SYSTEM TRAFFIC_Central (* System Configuration *)
  (* Standard: 61499-1 *)
  (* Version 0.4, 2009-03-05, JHC, Holobloc Inc., Deleted Application. *)
  (* Version 0.3, 2003-12-05, JHC, Rockwell Automation, Renamed from NEWSYSTEM. *)
  (* Version 0.2, 2002-11-05, JHC, Rockwell Automation, Fixed missing (empty) FBD in Application. *)
  (* Version 0.1, 2002-01-17, JHC, Rockwell Automation, Minor cleanup *)
  (* Version 0.0, 2000-05-27, JHC, Rockwell Automation *)
  DEVICE Device1 : FRAME_DEVICE(BOUNDS := [400,100,300,200], GRID := [1])
    RESOURCE VIEW1 : PANEL_RESOURCE(COLS := 1, ROWS := 6)
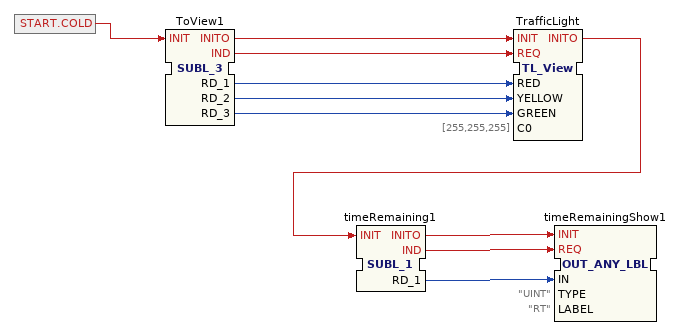
      FBS
        TrafficLight : TL_View(C0 := [255,255,255]);
        ToView1 : SUBL_3;
        timeRemaining1 : SUBL_1;
        timeRemainingShow1 : OUT_ANY_LBL(TYPE := "UINT", LABEL := "RT");
      END_FBS
      EVENT_CONNECTIONS
        START.COLD TO ToView1.INIT;
        ToView1.INITO TO TrafficLight.INIT;
        ToView1.IND TO TrafficLight.REQ;
        timeRemaining1.INITO TO timeRemainingShow1.INIT;
        timeRemaining1.IND TO timeRemainingShow1.REQ;
        TrafficLight.INITO TO timeRemaining1.INIT;
      END_CONNECTIONS
      DATA_CONNECTIONS
        ToView1.RD_1 TO TrafficLight.RED;
        ToView1.RD_2 TO TrafficLight.YELLOW;
        ToView1.RD_3 TO TrafficLight.GREEN;
        timeRemaining1.RD_1 TO timeRemainingShow1.IN;
      END_CONNECTIONS
    END_RESOURCE
    RESOURCE VIEW2 : PANEL_RESOURCE(COLS := 1, ROWS := 6)
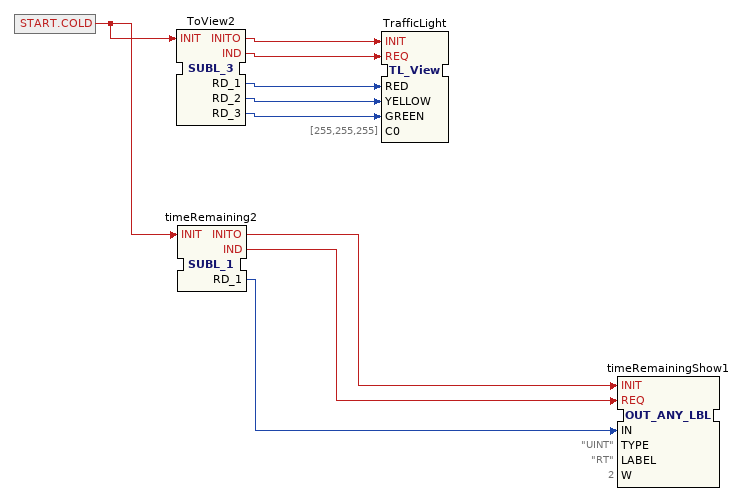
      FBS
        TrafficLight : TL_View(C0 := [255,255,255]);
        ToView2 : SUBL_3;
        timeRemaining2 : SUBL_1;
        timeRemainingShow1 : OUT_ANY_LBL(TYPE := "UINT", LABEL := "RT", W := 2);
      END_FBS
      EVENT_CONNECTIONS
        START.COLD TO ToView2.INIT;
        ToView2.INITO TO TrafficLight.INIT;
        ToView2.IND TO TrafficLight.REQ;
        START.COLD TO timeRemaining2.INIT;
        timeRemaining2.INITO TO timeRemainingShow1.INIT;
        timeRemaining2.IND TO timeRemainingShow1.REQ;
      END_CONNECTIONS
      DATA_CONNECTIONS
        ToView2.RD_1 TO TrafficLight.RED;
        ToView2.RD_2 TO TrafficLight.YELLOW;
        ToView2.RD_3 TO TrafficLight.GREEN;
        timeRemaining2.RD_1 TO timeRemainingShow1.IN;
      END_CONNECTIONS
    END_RESOURCE
    RESOURCE HMI : PANEL_RESOURCE(ROWS := 6, COLS := 1)
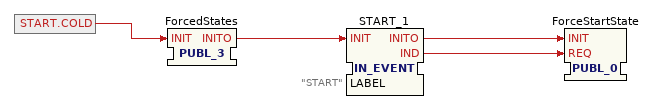
      FBS
        ForcedStates : PUBL_3;
        START_1 : IN_EVENT(LABEL := "START");
        ForceStartState : PUBL_0;
      END_FBS
      EVENT_CONNECTIONS
        ForcedStates.INITO TO START_1.INIT;
        START_1.INITO TO ForceStartState.INIT;
        START_1.IND TO ForceStartState.REQ;
        START.COLD TO ForcedStates.INIT;
      END_CONNECTIONS
    END_RESOURCE
    RESOURCE Model : EMB_RES
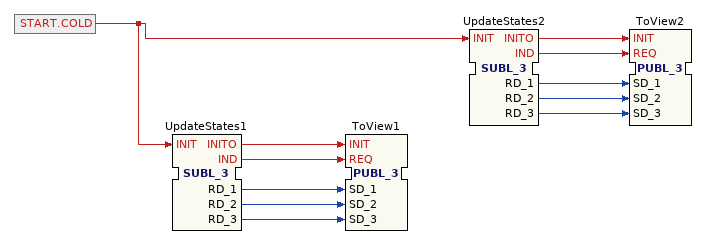
      FBS
        UpdateStates1 : SUBL_3;
        ToView1 : PUBL_3;
        ToView2 : PUBL_3;
        UpdateStates2 : SUBL_3;
      END_FBS
      EVENT_CONNECTIONS
        UpdateStates1.INITO TO ToView1.INIT;
        UpdateStates1.IND TO ToView1.REQ;
        UpdateStates2.INITO TO ToView2.INIT;
        UpdateStates2.IND TO ToView2.REQ;
        START.COLD TO UpdateStates1.INIT;
        START.COLD TO UpdateStates2.INIT;
      END_CONNECTIONS
      DATA_CONNECTIONS
        UpdateStates1.RD_1 TO ToView1.SD_1;
        UpdateStates1.RD_2 TO ToView1.SD_2;
        UpdateStates1.RD_3 TO ToView1.SD_3;
        UpdateStates2.RD_1 TO ToView2.SD_1;
        UpdateStates2.RD_2 TO ToView2.SD_2;
        UpdateStates2.RD_3 TO ToView2.SD_3;
      END_CONNECTIONS
    END_RESOURCE
    RESOURCE Control : EMB_RES
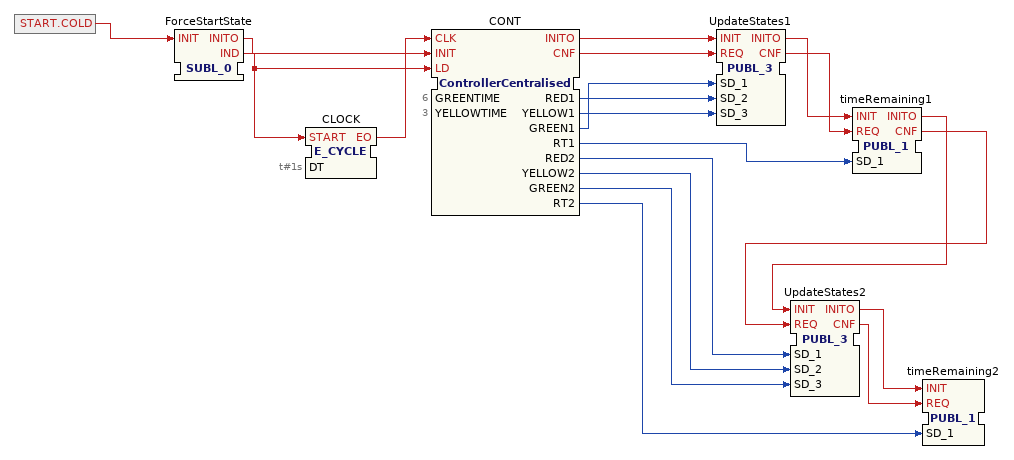
      FBS
        ForceStartState : SUBL_0;
        UpdateStates1 : PUBL_3;
        timeRemaining1 : PUBL_1;
        UpdateStates2 : PUBL_3;
        timeRemaining2 : PUBL_1;
        CONT : ControllerCentralised(GREENTIME := 6, YELLOWTIME := 3);
        CLOCK : E_CYCLE(DT := t#1s);
      END_FBS
      EVENT_CONNECTIONS
        START.COLD TO ForceStartState.INIT;
        UpdateStates1.INITO TO timeRemaining1.INIT;
        timeRemaining1.INITO TO UpdateStates2.INIT;
        UpdateStates2.INITO TO timeRemaining2.INIT;
        UpdateStates1.CNF TO timeRemaining1.REQ;
        UpdateStates2.CNF TO timeRemaining2.REQ;
        CLOCK.EO TO CONT.CLK;
        ForceStartState.INITO TO CONT.INIT;
        ForceStartState.IND TO CONT.LD;
        CONT.INITO TO UpdateStates1.INIT;
        CONT.CNF TO UpdateStates1.REQ;
        timeRemaining1.CNF TO UpdateStates2.REQ;
        ForceStartState.IND TO CLOCK.START;
      END_CONNECTIONS
      DATA_CONNECTIONS
        CONT.RED1 TO UpdateStates1.SD_1;
        CONT.YELLOW1 TO UpdateStates1.SD_2;
        CONT.GREEN1 TO UpdateStates1.SD_3;
        CONT.RT1 TO timeRemaining1.SD_1;
        CONT.RED2 TO UpdateStates2.SD_1;
        CONT.YELLOW2 TO UpdateStates2.SD_2;
        CONT.GREEN2 TO UpdateStates2.SD_3;
        CONT.RT2 TO timeRemaining2.SD_1;
      END_CONNECTIONS
    END_RESOURCE
  END_DEVICE
END_SYSTEM
